(* PLC project TestImplemetierung261220.project, CODESYS CODESYS V3.5 SP16 Patch 1 *)
(* stored: creationDateTime 2021-01-10T15:38:21.6544585, modificationDateTime 2021-01-10T15:37:56.945572 *)

PROGRAM PLC_PRG
  VAR
    rechner : calcFB;
  END_VAR

                    rechner.parameterA.name:='Parameter A';
rechner.parameterA.paramType:='Integer';
rechner.parameterA.required:=TRUE;
rechner.parameterB.name:='Parameter B';

rechner.parameterB.paramType:='Integer';
rechner.parameterB.required:=TRUE;

rechner();
(*manual parameter initalization*)




                  
END_PROGRAM

FUNCTION_BLOCK calcFB EXTENDS TJ.Skill_Template
  VAR_INPUT
    parameterA : TJ.SkillParameter := (default := 10, value := parameterA.default);
    parameterB : TJ.SkillParameter := (default := 10, value := parameterB.default);
  END_VAR
  VAR_OUTPUT
    result : INT;
  END_VAR

                    

(*Begin FB-Code*)
SUPER^(); (*extends Code of super-function-block*)



                  

METHOD execute : BOOL
                          THIS^.result:= THIS^.parameterA.value + THIS^.parameterB.value;

                        
END_METHOD

METHOD unsuspending : BOOL
                          
                        
END_METHOD

METHOD unholding : BOOL
                          
                        
END_METHOD

METHOD starting : BOOL
                          
                        
END_METHOD

METHOD resetting : BOOL
                          
                        
END_METHOD

METHOD suspending : BOOL
                          
                        
END_METHOD

METHOD stopping : BOOL
                          
                        
END_METHOD

METHOD holding : BOOL
                          
                        
END_METHOD

METHOD clearing : BOOL
                          
                        
END_METHOD

METHOD aborting : BOOL
                          
                        
END_METHOD

METHOD completing : BOOL
                          
                        
END_METHOD
END_FUNCTION_BLOCK

CONFIGURATION Device
  RESOURCE Application ON PLC
    TASK MainTask(INTERVAL := T#20ms, PRIORITY := 1);
    PROGRAM PLC_PRG WITH MainTask : PLC_PRG;
  END_RESOURCE
END_CONFIGURATION
